PROGRAM MAIN
VAR
	drive : AXIS_REF;
	
	fbMCReset : MC_Reset;
	fbMCPower : MC_Power;
	fbMCSetPosition : MC_SetPosition;
	
	bRun AT %Q* : BOOL := FALSE;
	bStarted : BOOL := FALSE;
	
	iTorqueOffset AT %Q* : INT := -3;
	iActualTorque AT %I* : INT;
	iActualTorqueConv : LREAL; // Nm
	iMaxRatedTorque : LREAL := 0.00768; // Nm
	
	iMaxVel : INT  := 300;
	iMaxPos : REAL := 182;
	iMinPos : REAL := 005;
END_VAR

drive.ReadStatus();
fbMCSetPosition(Axis:=drive, Execute:=TRUE, Position:=0);

iActualTorqueConv := INT_TO_LREAL(iActualTorque) / 1000 * iMaxRatedTorque;

IF ABS(drive.NcToPlc.ActVelo) > iMaxVel THEN
	bRun := FALSE;
END_IF

IF NOT bStarted THEN
	fbMCReset(Axis:=drive);
	fbMCPower(Axis:=drive, Enable:= TRUE, Enable_Positive:=TRUE, Enable_Negative:=TRUE);
	// if motor powered, set to started
	IF fbMCPower.Status THEN
		bStarted := TRUE;
	END_IF
ELSE
	iMaxVel := iMaxVel; // pass statement
END_IF

END_PROGRAM

(* stored: Version 1.1.0.1, ProductVersion 3.1.4024.13
   POU MAIN: Id {13a96fbb-10e3-44e8-a51b-e00ae15eb7c3}, SpecialFunc None *)
